(* FB_TankFourCompartments contain 4 SingleTank
*)
FUNCTION_BLOCK FB_TankFourCompartments
VAR
	sName : STRING;
	lrWeight : LREAL;				//Total Weight of the 4 tanks
	sWeightUnit : STRING := 'Kg'; 	// Kg
	fbTank1 : FB_SingleTankV0;
	fbTank2 : FB_SingleTankV0;
	fbTank3 : FB_SingleTankV0;
	fbTank4 : FB_SingleTankV0;
	
	bAllowInMaterial : BOOL;
	bAllowOutMaterial : BOOL;
	lrLimitMinWeight : LREAL;
	lrLimitMaxWeight : LREAL;
	lrWeightWithdraw : LREAL; 		// weight withdraw Request 
	bEnoughWithdraw : BOOL;
END_VAR

fbTank1();
fbTank2();
fbTank3();
fbTank4();
bAllowInMaterial := lrWeight < lrLimitMaxWeight;	
bAllowOutMaterial := lrWeight > lrLimitMinWeight;
bEnoughWithdraw := lrWeight > (lrWeightWithdraw + lrLimitMinWeight);

PROPERTY AllowIn : Reference to bool
GET
AllowIn ref= bAllowInMaterial;
END_GET
END_PROPERTY

(*
| Check the minimum condition  (lrWeight > lrLimitMinWeight
								AND piLslow.In;)
*)
PROPERTY AllowOut : REFERENCE TO BOOL
GET
AllowOut ref= bAllowOutMaterial;
END_GET
END_PROPERTY

(*
|Check every single tank enough weight to withdraw
|I'm not sure whether this function CLEAN ? SOLID principle
*)
PROPERTY EnoughWithdraw : reference to bool
GET
EnoughWithdraw ref= bEnoughWithdraw;
END_GET
END_PROPERTY

METHOD FirstCycle : BOOL
VAR_INPUT
	sName : STRING;
	sWeightUnit : STRING;
END_VAR
THIS^.sName := sName;
THIS^.sWeightUnit := sWeightUnit;

fbTank1.Name := CONCAT(sName, ' part 1');
fbTank1.WeightUnit := sWeightUnit;

fbTank2.Name := CONCAT(sName, ' part 2');
fbTank2.WeightUnit := sWeightUnit;

fbTank3.Name := CONCAT(sName, ' part 3');
fbTank3.WeightUnit := sWeightUnit;

fbTank4.Name := CONCAT(sName, ' part 4');
fbTank4.WeightUnit := sWeightUnit;
END_METHOD

PROPERTY LimitMaxWeight : lreal
GET
LimitMaxWeight := lrLimitMaxWeight;
END_GET
SET
lrLimitMaxWeight := LimitMaxWeight;
END_SET
END_PROPERTY

PROPERTY LimitMinWeight : lreal
GET
LimitMinWeight := lrLimitMinWeight;
END_GET
SET
lrLimitMinWeight := LimitMinWeight;
END_SET
END_PROPERTY

PROPERTY Name : String
GET
Name := sName;
END_GET
SET
sName := Name;
END_SET
END_PROPERTY

PROPERTY Ref_Tank1 : Reference to FB_SingleTankV0
GET
Ref_Tank1 ref= fbTank1;
END_GET
END_PROPERTY

PROPERTY Ref_Tank2 : Reference to FB_SingleTankV0
GET
Ref_Tank2 ref= fbTank2;
END_GET
END_PROPERTY

PROPERTY Ref_Tank3 : Reference to FB_SingleTankV0
GET
Ref_Tank3 ref= fbTank3;
END_GET
END_PROPERTY

PROPERTY Ref_Tank4 : Reference to FB_SingleTankV0
GET
Ref_Tank4 ref= fbTank4;
END_GET
END_PROPERTY

PROPERTY Weight : lreal
GET
Weight := lrWeight;
END_GET
SET
lrWeight := Weight;
END_SET
END_PROPERTY

PROPERTY WeightUnit : string
GET
WeightUnit := sWeightUnit;
END_GET
SET
sWeightUnit := WeightUnit;
END_SET
END_PROPERTY

PROPERTY WeightWithdraw : lreal
GET
WeightWithdraw := lrWeightWithdraw;
END_GET
SET
lrWeightWithdraw := WeightWithdraw;
END_SET
END_PROPERTY

END_FUNCTION_BLOCK

(* stored: Version 1.1.0.1, ProductVersion 3.1.4024.12
   POU FB_TankFourCompartments: Id {c9822f20-c949-4c54-bd7b-9d89bf59690c}, SpecialFunc None
   Property AllowIn: Id {d64b247e-5b5d-4e76-8d58-f3f9586a9da0}
   Get Get: Id {fb0a8198-73d2-4fe2-ae8c-01950aad06e5}
   Property AllowOut: Id {f5ad63cd-639d-4454-94ab-652011eb22de}
   Get Get: Id {2a9a67aa-d4e7-46df-9388-5ae765f1da4d}
   Property EnoughWithdraw: Id {53e63e81-c0ca-44a8-9900-22a7b14f8cdc}
   Get Get: Id {c5b3a758-c913-43f0-8bec-5194aa638d4d}
   Method FirstCycle: Id {7d733376-fb1c-432c-b6b7-4a1960c67340}
   Property LimitMaxWeight: Id {b59d8be2-d633-4a6d-9c4c-27551b4f04e8}
   Get Get: Id {01157412-39dd-4149-8eeb-406729f6f0aa}
   Set Set: Id {f10dc189-f270-424e-bf74-0bf16c3fd33a}
   Property LimitMinWeight: Id {004677b0-17d6-48c1-832f-cf1a0ebf3f3a}
   Get Get: Id {19f9ff2c-3fc9-44dc-a6ff-1ffec7be245b}
   Set Set: Id {f5e73618-addc-4579-85da-2ba14a5c7f7a}
   Property Name: Id {14bcf70a-e2fd-4276-afc1-d57e39cdc948}
   Get Get: Id {bce301fd-0189-48a5-a654-040e4d1faee3}
   Set Set: Id {a8e8bcc4-57e1-4aac-8638-d4af2b02ac9b}
   Property Ref_Tank1: Id {470d455d-9798-416b-b527-82f70c0f0525}
   Get Get: Id {39ae51a8-910c-410d-8f6a-d9edd810cf9c}
   Property Ref_Tank2: Id {73998b37-398a-401c-8f1d-7d57ced4191f}
   Get Get: Id {e410b360-6b34-44fd-b19f-de3f9a6f10ac}
   Property Ref_Tank3: Id {86df6bbe-af79-4315-a793-c90d3e1ec793}
   Get Get: Id {7b91788c-1481-401b-a3ee-3fde064b710a}
   Property Ref_Tank4: Id {7bcf008e-1a49-4f12-8f39-e7665a8d8a1d}
   Get Get: Id {f86475f3-8691-4d38-8631-d097c6191c56}
   Property Weight: Id {41eb71b2-11cc-4774-bd88-15f3cb53eba1}
   Get Get: Id {319b6d1d-de23-4a36-9999-2455b72c41c2}
   Set Set: Id {8006daec-6c4f-4e49-8925-7b140cb09b7b}
   Property WeightUnit: Id {71bda2f2-a61e-40f2-a8f8-c1b481bec1cf}
   Get Get: Id {8fc1816b-737c-4924-974b-fc70f557c29b}
   Set Set: Id {db357657-ef56-4cb6-a9ac-27018747b80b}
   Property WeightWithdraw: Id {04258af5-bb97-4da9-a61e-e99ef96c825e}
   Get Get: Id {99258e5a-1cf5-448d-b7f2-76cfb8ad1d70}
   Set Set: Id {eea76fa7-c0ae-4c50-b2fa-c3b4a440368d} *)
